{attribute 'qualified_only'}
{attribute 'strict'}
TYPE E_SignalTowerLampMode :
(
	Disable := 0,
	AlwaysOn,
	Flash_05Hz,
	Flash_1Hz,
	Flash_2Hz
)DINT;
END_TYPE

(* stored: Version 1.1.0.1, ProductVersion 3.1.4024.13
   DUT E_SignalTowerLampMode: Id {d42bc509-d420-48ef-89b8-b545d09f76c0} *)
